DATA_BLOCK "Temperatur_DB"
{ S7_Optimized_Access := 'TRUE' }
VERSION : 0.1
NON_RETAIN
"Temperatur"

BEGIN

END_DATA_BLOCK

